// TIA Portal V19 export
DATA_BLOCK "ProfileMng"   // DB19
// stored: InstanceOfName ProgramsManager_FB, InstanceOfType FB
"ProgramsManager_FB"
   // VAR_INPUT
   //    ArchiveNo : USInt;
   //    Enable : Bool;
   //    RstAlarms : Bool;
   // END_VAR
   // VAR_OUTPUT
   //    COut : Struct
   //       AlarmsPresence : Bool;
   //       WarningPresence : Bool;
   //       ProgramUpdated : Bool;
   //    END_STRUCT;
   //    Warning : Struct
   //       Scada_WrongPrgNo : Bool;
   //       Scada_WrongPivotTable : Bool;
   //       Scada_ArchiveFull : Bool;
   //       Scada_ReadArchiveError : Bool;
   //       Scada_WriteArchiveError : Bool;
   //    END_STRUCT;
   // END_VAR
   // VAR_IN_OUT
   //    PIVOT : Array[*] of "Prg_Pivot";
   //    GET_ITF : "Prg_GetITF";
   //    RWD_EMPTY : Variant;
   //    RWD_UPDATE : Variant;
   //    RWD_GET : Variant;
   //    RWD_HMI : Variant;
   //    RWD_SCADA : Variant;
   //    RWDHeader_HMI : "Prg_Header";
   //    RWDHeader_SCADA : "Prg_Header";
   //    HMI : "Prg_HMI";
   //    SCADA : "Prg_SCADA";
   // END_VAR
   // VAR
   //    Status : Int;
   //    Sts : Struct
   //       ReadDone : Bool;
   //       ReadError : Bool;
   //       WriteDone : Bool;
   //       WriteError : Bool;
   //       PivotRecordRW : Int;
   //       PivotIndexRW : Int;
   //       PivotRecordFirstFree : Int;
   //       PivotIndexRecordFirstFree : Int;
   //       RecordToWrite : Int;
   //       IndexToUpdate : Int;
   //       ListFirstIndex : Int;
   //       ListIndexMin : Int;
   //       ListIndexMax : Int;
   //       ProgramNumberToManage : DInt;
   //       PercentageUnitVal : Real;
   //       ScadaOpBusy : Bool;
   //       ProgramUpdated : Bool;
   //    END_STRUCT;
   //    Ctrl : Struct
   //       ReadExe : Bool;
   //       WriteExe : Bool;
   //    END_STRUCT;
   //    Get : Struct
   //       Status : Int;
   //       RecordNo : Int;
   //       ExeRead : Bool;
   //    END_STRUCT;
   //    Msg : Struct
   //       Scada_WrongPrgNo : Bool;
   //       Scada_WrongPivotTable : Bool;
   //       Scada_ArchiveFull : Bool;
   //       Scada_ReadArchiveError : Bool;
   //       Scada_WriteArchiveError : Bool;
   //    END_STRUCT;
   //    SortPivotTable : "SortPivot";
   //    tonDone : IEC_TIMER;
   //    tonSaveDoneScada : IEC_TIMER;
   //    tonDeleteDoneScada : IEC_TIMER;
   //    tonReadDoneScada : IEC_TIMER;
   //    tonCopyDelay : IEC_TIMER;
   // END_VAR
BEGIN
END_DATA_BLOCK
